//structure to configure how messages are built
TYPE ST_ConfigMsgBuild :
STRUCT
  AlarmMsg          : ST_ShowMsgFields;
  InfoMsg           : ST_ShowMsgFields;
  RegisterMsg       : ST_ShowMsgFields;
  bShowRegisterMsg  : BOOL := FALSE;
END_STRUCT
END_TYPE

(* stored: Version 1.1.0.1, ProductVersion 3.1.4024.12
   DUT ST_ConfigMsgBuild: Id {1e03d47f-f01a-40c3-b81e-d7f7d0a36546} *)
